(* CoDeSys 2.3 export: MANUAL_CARRITOS.EXP *)

(* POU Manual/Manual_Carritos, LD *)
PROGRAM Manual_Carritos
VAR

END_VAR
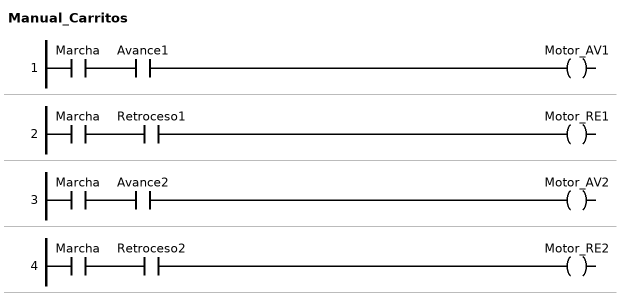
_LD_ (* Ladder Diagram *)
NETWORK 1
	[Marcha] - [Avance1] --- (Motor_AV1)
NETWORK 2
	[Marcha] - [Retroceso1] --- (Motor_RE1)
NETWORK 3
	[Marcha] - [Avance2] --- (Motor_AV2)
NETWORK 4
	[Marcha] - [Retroceso2] --- (Motor_RE2)
_END_LD_
(* the same logic as Structured Text *)
(* Network 1 *)
Motor_AV1 := Marcha AND Avance1;
(* Network 2 *)
Motor_RE1 := Marcha AND Retroceso1;
(* Network 3 *)
Motor_AV2 := Marcha AND Avance2;
(* Network 4 *)
Motor_RE2 := Marcha AND Retroceso2;
END_PROGRAM
